TYPE E_ProductFlowState :
(
	none := 0,
	busy,
	done,
	error
);
END_TYPE

(* stored: Version 1.1.0.1, ProductVersion 3.1.0.19
   DUT E_ProductFlowState: Id {f1b374a5-05e8-4973-847a-3a7ff6103401} *)
